SYSTEM Test Big Computation ser 10
  (* Version 1.0, 2005-12-23, Goran Cengic, Chalmers *)
  DEVICE Test Device : DeviceType_not_used
    RESOURCE Test Resource : ResourceType_not_used
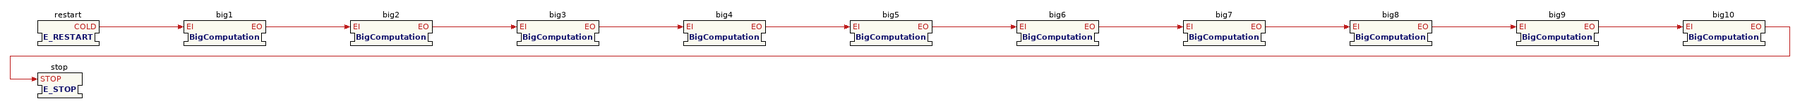
      FBS
        restart : E_RESTART;
        stop : E_STOP;
        big1 : BigComputation;
        big2 : BigComputation;
        big3 : BigComputation;
        big4 : BigComputation;
        big5 : BigComputation;
        big6 : BigComputation;
        big7 : BigComputation;
        big8 : BigComputation;
        big9 : BigComputation;
        big10 : BigComputation;
      END_FBS
      EVENT_CONNECTIONS
        restart.COLD TO big1.EI;
        big1.EO TO big2.EI;
        big2.EO TO big3.EI;
        big3.EO TO big4.EI;
        big4.EO TO big5.EI;
        big5.EO TO big6.EI;
        big6.EO TO big7.EI;
        big7.EO TO big8.EI;
        big8.EO TO big9.EI;
        big9.EO TO big10.EI;
        big10.EO TO stop.STOP;
      END_CONNECTIONS
    END_RESOURCE
  END_DEVICE
END_SYSTEM
